// TIA Portal V20 export
FUNCTION "PostProcessing" : Void   // FC57, LAD
TITLE = Post Processing
// V1.0  25.05.04  Safety test program: sending data via F-link
// stored: Namespace Safety, SetENOAutomatically false
BEGIN

REGION Network 1: Sending data to BA010, ReelCut #1
   // V1.0  25.05.04  Safety test program: FlinkSendToBA10AC1
   //                 Send ID: 102, Receive ID: 103
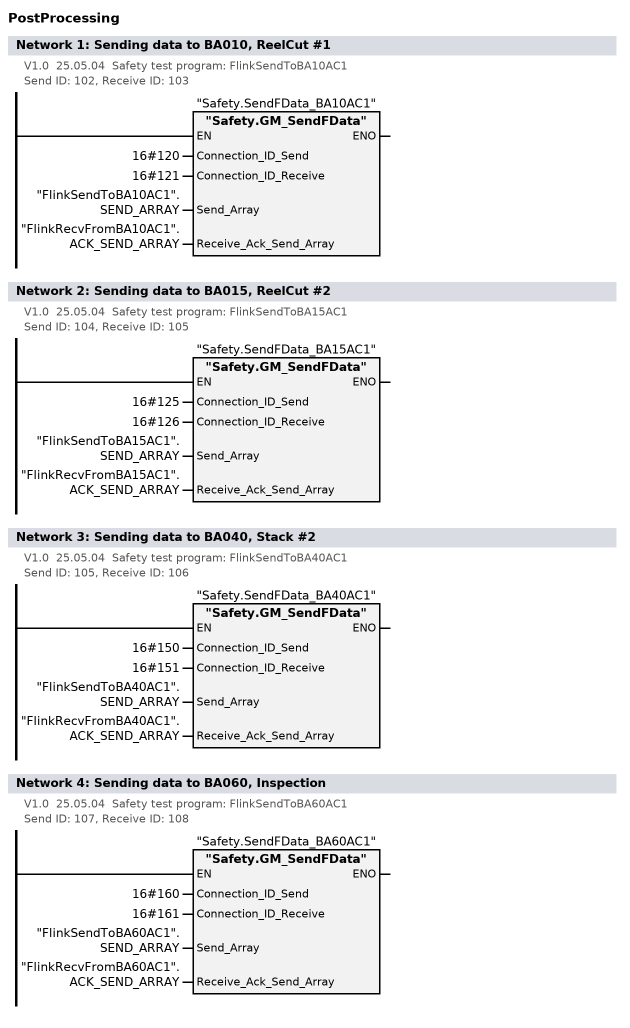
   RUNG wire#powerrail
      "Safety.SendFData_BA10AC1"(Connection_ID_Send := 16#120, Connection_ID_Receive := 16#121, Send_Array := "FlinkSendToBA10AC1".SEND_ARRAY, Receive_Ack_Send_Array := "FlinkRecvFromBA10AC1".ACK_SEND_ARRAY)
   END_RUNG
   // the same network as SCL:
   "Safety.SendFData_BA10AC1"(Connection_ID_Send := 16#120,   // "Safety.GM_SendFData"
                           Connection_ID_Receive := 16#121,
                           Send_Array := "FlinkSendToBA10AC1".SEND_ARRAY,
                           Receive_Ack_Send_Array := "FlinkRecvFromBA10AC1".ACK_SEND_ARRAY);
END_REGION

REGION Network 2: Sending data to BA015, ReelCut #2
   // V1.0  25.05.04  Safety test program: FlinkSendToBA15AC1
   //                 Send ID: 104, Receive ID: 105
   RUNG wire#powerrail
      "Safety.SendFData_BA15AC1"(Connection_ID_Send := 16#125, Connection_ID_Receive := 16#126, Send_Array := "FlinkSendToBA15AC1".SEND_ARRAY, Receive_Ack_Send_Array := "FlinkRecvFromBA15AC1".ACK_SEND_ARRAY)
   END_RUNG
   // the same network as SCL:
   "Safety.SendFData_BA15AC1"(Connection_ID_Send := 16#125,   // "Safety.GM_SendFData"
                           Connection_ID_Receive := 16#126,
                           Send_Array := "FlinkSendToBA15AC1".SEND_ARRAY,
                           Receive_Ack_Send_Array := "FlinkRecvFromBA15AC1".ACK_SEND_ARRAY);
END_REGION

REGION Network 3: Sending data to BA040, Stack #2
   // V1.0  25.05.04  Safety test program: FlinkSendToBA40AC1
   //                 Send ID: 105, Receive ID: 106
   RUNG wire#powerrail
      "Safety.SendFData_BA40AC1"(Connection_ID_Send := 16#150, Connection_ID_Receive := 16#151, Send_Array := "FlinkSendToBA40AC1".SEND_ARRAY, Receive_Ack_Send_Array := "FlinkRecvFromBA40AC1".ACK_SEND_ARRAY)
   END_RUNG
   // the same network as SCL:
   "Safety.SendFData_BA40AC1"(Connection_ID_Send := 16#150,   // "Safety.GM_SendFData"
                           Connection_ID_Receive := 16#151,
                           Send_Array := "FlinkSendToBA40AC1".SEND_ARRAY,
                           Receive_Ack_Send_Array := "FlinkRecvFromBA40AC1".ACK_SEND_ARRAY);
END_REGION

REGION Network 4: Sending data to BA060, Inspection
   // V1.0  25.05.04  Safety test program: FlinkSendToBA60AC1
   //                 Send ID: 107, Receive ID: 108
   RUNG wire#powerrail
      "Safety.SendFData_BA60AC1"(Connection_ID_Send := 16#160, Connection_ID_Receive := 16#161, Send_Array := "FlinkSendToBA60AC1".SEND_ARRAY, Receive_Ack_Send_Array := "FlinkRecvFromBA60AC1".ACK_SEND_ARRAY)
   END_RUNG
   // the same network as SCL:
   "Safety.SendFData_BA60AC1"(Connection_ID_Send := 16#160,   // "Safety.GM_SendFData"
                           Connection_ID_Receive := 16#161,
                           Send_Array := "FlinkSendToBA60AC1".SEND_ARRAY,
                           Receive_Ack_Send_Array := "FlinkRecvFromBA60AC1".ACK_SEND_ARRAY);
END_REGION

REGION Network 5 (SCL): Set ACK_OP value in DataToSafety
   "Safety.DataToSafety".ackSafetyFromHmi := "Safety.DataFromStandard".ackSafetyFromHmi;
   "Safety.DataFromSafety".ackOP_changeRequired := "Safety.InstMain_Safety_RTG1".instAckOP.Q;
END_REGION
END_FUNCTION
